// TIA Portal V15.1 export
// export: Created 2024-05-17T05:38:12.5998279Z, ExportSetting WithDefaults, DisplayName Totally Integrated Automation Portal, DisplayVersion V15.1 Update 5, DisplayName TIA Portal Openness, DisplayVersion V15.1 Update 5, DisplayName SINAMICS Startdrive Advanced, DisplayVersion V15.1, DisplayName G130, G150, S120, S150, SINAMICS MV, S210, DisplayVersion V15.1, DisplayName G110M, G120, G120C, G120D, G120P, DisplayVersion V15.1, DisplayName STEP 7 Professional, DisplayVersion V15.1 Update 5, DisplayName STEP 7 Safety, DisplayVersion V15.1, DisplayName WinCC Professional, DisplayVersion V15.1 Update 5, DisplayName SIMATIC Visualization Architect, DisplayVersion V15.1
DATA_BLOCK "_INTLK"   // DB20
{ S7_Optimized_Access := 'FALSE' }
AUTHOR : VCC
NAME : INTLDB
VERSION : 0.1
// stored: AutoNumber false, DBAccessibleFromOPCUA true, IsOnlyStoredInLoadMemory false, IsWriteProtectedInAS false
   VAR RETAIN
      _209210ZMS011BypassSC { ExternalAccessible := 'False'; ExternalVisible := 'False'; ExternalWritable := 'False'} : Bool;   // StartCondition Bypass sub modezone 210ZMS011 / StartCondition Bypass modezone MZ1
      _209210ZMS011SimPartSC { ExternalAccessible := 'False'; ExternalVisible := 'False'; ExternalWritable := 'False'} : Bool;   // StartCondition Simulation with part sub modezone 210ZMS011 / StartCondition Simulation with part modezone MZ1
      _209210ZMS011SimNoPartSC { ExternalAccessible := 'False'; ExternalVisible := 'False'; ExternalWritable := 'False'} : Bool;   // StartCondition Simulation without part sub modezone 210ZMS011 / StartCondition Simulation without part modezone MZ1
      _209210ZMS011MaintSC { ExternalAccessible := 'False'; ExternalVisible := 'False'; ExternalWritable := 'False'} : Bool;   // StartCondition Maintenance sub modezone 210ZMS011 / StartCondition Maintenance modezone MZ1
      _209210ZMS011HomerunSC { ExternalAccessible := 'False'; ExternalVisible := 'False'; ExternalWritable := 'False'} : Bool;   // StartCondition Homerun sub modezone 210ZMS011 / StartCondition Homerun modezone MZ1
      _209210ZMS012BypassSC { ExternalAccessible := 'False'; ExternalVisible := 'False'; ExternalWritable := 'False'} : Bool;   // StartCondition Bypass sub modezone 210ZMS012 / StartCondition Bypass modezone MZ1
      _209210ZMS012SimPartSC { ExternalAccessible := 'False'; ExternalVisible := 'False'; ExternalWritable := 'False'} : Bool;   // StartCondition Simulation with part sub modezone 210ZMS012 / StartCondition Simulation with part modezone MZ1
      _209210ZMS012SimNoPartSC { ExternalAccessible := 'False'; ExternalVisible := 'False'; ExternalWritable := 'False'} : Bool;   // StartCondition Simulation without part sub modezone 210ZMS012 / StartCondition Simulation without part modezone MZ1
      _209210ZMS012MaintSC { ExternalAccessible := 'False'; ExternalVisible := 'False'; ExternalWritable := 'False'} : Bool;   // StartCondition Maintenance sub modezone 210ZMS012 / StartCondition Maintenance modezone MZ1
      _209210ZMS012HomerunSC { ExternalAccessible := 'False'; ExternalVisible := 'False'; ExternalWritable := 'False'} : Bool;   // StartCondition Homerun sub modezone 210ZMS012 / StartCondition Homerun modezone MZ1
      _209210ZMS013BypassSC { ExternalAccessible := 'False'; ExternalVisible := 'False'; ExternalWritable := 'False'} : Bool;   // StartCondition Bypass sub modezone 210ZMS013 / StartCondition Bypass modezone MZ1
      _209210ZMS013SimPartSC { ExternalAccessible := 'False'; ExternalVisible := 'False'; ExternalWritable := 'False'} : Bool;   // StartCondition Simulation with part sub modezone 210ZMS013 / StartCondition Simulation with part modezone MZ1
      _209210ZMS013SimNoPartSC { ExternalAccessible := 'False'; ExternalVisible := 'False'; ExternalWritable := 'False'} : Bool;   // StartCondition Simulation without part sub modezone 210ZMS013 / StartCondition Simulation without part modezone MZ1
      _209210ZMS013MaintSC { ExternalAccessible := 'False'; ExternalVisible := 'False'; ExternalWritable := 'False'} : Bool;   // StartCondition Maintenance sub modezone 210ZMS013 / StartCondition Maintenance modezone MZ1
      _209210ZMS013HomerunSC { ExternalAccessible := 'False'; ExternalVisible := 'False'; ExternalWritable := 'False'} : Bool;   // StartCondition Homerun sub modezone 210ZMS013 / StartCondition Homerun modezone MZ1
      _209220ZMS011BypassSC { ExternalAccessible := 'False'; ExternalVisible := 'False'; ExternalWritable := 'False'} : Bool;   // StartCondition Bypass sub modezone 220ZMS011 / StartCondition Bypass modezone MZ1
      _209220ZMS011SimPartSC { ExternalAccessible := 'False'; ExternalVisible := 'False'; ExternalWritable := 'False'} : Bool;   // StartCondition Simulation with part sub modezone 220ZMS011 / StartCondition Simulation with part modezone MZ1
      _209220ZMS011SimNoPartSC { ExternalAccessible := 'False'; ExternalVisible := 'False'; ExternalWritable := 'False'} : Bool;   // StartCondition Simulation without part sub modezone 220ZMS011 / StartCondition Simulation without part modezone MZ1
      _209220ZMS011MaintSC { ExternalAccessible := 'False'; ExternalVisible := 'False'; ExternalWritable := 'False'} : Bool;   // StartCondition Maintenance sub modezone 220ZMS011 / StartCondition Maintenance modezone MZ1
      _209220ZMS011HomerunSC { ExternalAccessible := 'False'; ExternalVisible := 'False'; ExternalWritable := 'False'} : Bool;   // StartCondition Homerun sub modezone 220ZMS011 / StartCondition Homerun modezone MZ1
      _209220ZMS012BypassSC { ExternalAccessible := 'False'; ExternalVisible := 'False'; ExternalWritable := 'False'} : Bool;   // StartCondition Bypass sub modezone 220ZMS012 / StartCondition Bypass modezone MZ1
      _209220ZMS012SimPartSC { ExternalAccessible := 'False'; ExternalVisible := 'False'; ExternalWritable := 'False'} : Bool;   // StartCondition Simulation with part sub modezone 220ZMS012 / StartCondition Simulation with part modezone MZ1
      _209220ZMS012SimNoPartSC { ExternalAccessible := 'False'; ExternalVisible := 'False'; ExternalWritable := 'False'} : Bool;   // StartCondition Simulation without part sub modezone 220ZMS012 / StartCondition Simulation without part modezone MZ1
      _209220ZMS012MaintSC { ExternalAccessible := 'False'; ExternalVisible := 'False'; ExternalWritable := 'False'} : Bool;   // StartCondition Maintenance sub modezone 220ZMS012 / StartCondition Maintenance modezone MZ1
      _209220ZMS012HomerunSC { ExternalAccessible := 'False'; ExternalVisible := 'False'; ExternalWritable := 'False'} : Bool;   // StartCondition Homerun sub modezone 220ZMS012 / StartCondition Homerun modezone MZ1
      _209220ZMS013BypassSC { ExternalAccessible := 'False'; ExternalVisible := 'False'; ExternalWritable := 'False'} : Bool;   // StartCondition Bypass sub modezone 220ZMS013 / StartCondition Bypass modezone MZ1
      _209220ZMS013SimPartSC { ExternalAccessible := 'False'; ExternalVisible := 'False'; ExternalWritable := 'False'} : Bool;   // StartCondition Simulation with part sub modezone 220ZMS013 / StartCondition Simulation with part modezone MZ1
      _209220ZMS013SimNoPartSC { ExternalAccessible := 'False'; ExternalVisible := 'False'; ExternalWritable := 'False'} : Bool;   // StartCondition Simulation without part sub modezone 220ZMS013 / StartCondition Simulation without part modezone MZ1
      _209220ZMS013MaintSC { ExternalAccessible := 'False'; ExternalVisible := 'False'; ExternalWritable := 'False'} : Bool;   // StartCondition Maintenance sub modezone 220ZMS013 / StartCondition Maintenance modezone MZ1
      _209220ZMS013HomerunSC { ExternalAccessible := 'False'; ExternalVisible := 'False'; ExternalWritable := 'False'} : Bool;   // StartCondition Homerun sub modezone 220ZMS013 / StartCondition Homerun modezone MZ1
      _209230ZM01BypassSC { ExternalAccessible := 'False'; ExternalVisible := 'False'; ExternalWritable := 'False'} : Bool;   // StartCondition Bypass sub modezone 230ZM01 / StartCondition Bypass modezone MZ1
      _209230ZM01SimPartSC { ExternalAccessible := 'False'; ExternalVisible := 'False'; ExternalWritable := 'False'} : Bool;   // StartCondition Simulation with part sub modezone 230ZM01 / StartCondition Simulation with part modezone MZ1
      _209230ZM01SimNoPartSC { ExternalAccessible := 'False'; ExternalVisible := 'False'; ExternalWritable := 'False'} : Bool;   // StartCondition Simulation without part sub modezone 230ZM01 / StartCondition Simulation without part modezone MZ1
      _209230ZM01MaintSC { ExternalAccessible := 'False'; ExternalVisible := 'False'; ExternalWritable := 'False'} : Bool;   // StartCondition Maintenance sub modezone 230ZM01 / StartCondition Maintenance modezone MZ1
      _209230ZM01HomerunSC { ExternalAccessible := 'False'; ExternalVisible := 'False'; ExternalWritable := 'False'} : Bool;   // StartCondition Homerun sub modezone 230ZM01 / StartCondition Homerun modezone MZ1
   END_VAR
BEGIN
END_DATA_BLOCK
